FUNCTION_BLOCK FB_AlarmControler EXTENDS FB_VisuEventsHandling IMPLEMENTS I_AlarmControler
VAR
	sName 					: STRING;					(*  *)

	bInit 					: BOOL;						(*  *)
	bAbort 					: BOOL;						(*  *)
	bClear					: BOOL;						(*  *)
	bClearAll 				: BOOL;						(*  *)
	bConfirm 				: BOOL;						(*  *)
	bConfirmAll 			: BOOL;						(*  *)
	bExport 				: BOOL;						(*  *)
	
	bResetConfirmation 		: BOOL;						(*  *)
	sFileName				: STRING;					(*  *)
	
	bActive 				: BOOL;						(*  *)
	bBusy					: BOOL;						(*  *)
	bError					: BOOL;						(*  *)
	iErrorID 				: HRESULT;					(*  *)
	iResult					: HRESULT;					(*  *)
	eAlarmControlerState 	: E_AlarmControlerState;	(*  *)
	
	ipFilter 				: I_TcEventFilter;			(*  *)
	fbEventLogger 			: FB_TcEventLogger;			(*  *)
END_VAR

(* Execute parent logic *)
SUPER^();

(* Run main state machine *)
StateMachine();

PROPERTY Active : REFERENCE TO BOOL
GET
Active REF= bActive;
END_GET
END_PROPERTY

PROPERTY ActiveCritical : REFERENCE TO UDINT
GET
ActiveCritical REF= iActiveCritical;
END_GET
END_PROPERTY

PROPERTY ActiveError : REFERENCE TO UDINT
GET
ActiveError REF= iActiveError;
END_GET
END_PROPERTY

PROPERTY ActiveInfo : REFERENCE TO UDINT
GET
ActiveInfo REF= iActiveInfo;
END_GET
END_PROPERTY

PROPERTY ActiveVerbose : REFERENCE TO UDINT
GET
ActiveVerbose REF= iActiveVerbose;
END_GET
END_PROPERTY

PROPERTY ActiveWarrning : REFERENCE TO UDINT
GET
ActiveWarrning REF= iActiveWarning;
END_GET
END_PROPERTY

PROPERTY AlarmsTable : REFERENCE TO ARRAY[1..iMAX_EVENTS] OF ST_Event
GET
AlarmsTable REF= arrActiveAlarms;
END_GET
END_PROPERTY

PROPERTY Busy : REFERENCE TO BOOL
GET
Busy REF= bBusy;
END_GET
END_PROPERTY

PROPERTY Error : REFERENCE TO BOOL
GET
Error REF= bError;
END_GET
END_PROPERTY

PROPERTY ErrorID : REFERENCE TO HRESULT
GET
ErrorID REF= iResult;
END_GET
END_PROPERTY

PROPERTY EventsTable : REFERENCE TO ARRAY[1..iMAX_EVENTS] OF ST_Event
GET
EventsTable REF= arrEvents;
END_GET
END_PROPERTY

PROPERTY FileName : STRING
GET
FileName := sFileName;
END_GET
SET
sFileName := FileName;
END_SET
END_PROPERTY

PROPERTY MaxEvents : UDINT
GET
MaxEvents := iMAX_EVENTS;
END_GET
END_PROPERTY

METHOD MR_Abort : BOOL
VAR_INPUT
END_VAR
IF eAlarmControlerState > ALARM_CONTROLER_UNINITIALIZED THEN
	bAbort := TRUE;
	MR_Abort := FALSE;
	bBusy := TRUE;
	
	eAlarmControlerState := ALARM_CONTROLER_ABORTING;
	fbMachineLogger.MR_AddLogs(CONCAT(sName,' : abort requested'));	
	
ELSIF eAlarmControlerState = ALARM_CONTROLER_UNINITIALIZED THEN
	bAbort := FALSE;
	MR_Abort := TRUE;
	bBusy := FALSE;
	bActive := FALSE;
	
	fbMachineLogger.MR_AddLogs(CONCAT(sName,' : abort done'));	
	
END_IF
END_METHOD

METHOD MR_Clear : BOOL
VAR_INPUT
	ipFilter : I_TcEventFilter;
	bResetConfirmation : BOOL;
END_VAR
IF eAlarmControlerState = ALARM_CONTROLER_IDLE THEN
	bClear := TRUE;
	MR_Clear := FALSE;
	bBusy := TRUE;
	THIS^.ipFilter := ipFilter;
	THIS^.bResetConfirmation := bResetConfirmation;
	
	eAlarmControlerState := ALARM_CONTROLER_CLEAR;
	fbMachineLogger.MR_AddLogs(CONCAT(sName,' : clear requested'));		
	
ELSIF eAlarmControlerState = ALARM_CONTROLER_CLEAR_DONE THEN
	bClear := FALSE;
	MR_Clear := TRUE;	
	bBusy := FALSE;
	
	fbMachineLogger.MR_AddLogs(CONCAT(sName,' : clear done'));		
	
END_IF
END_METHOD

METHOD MR_ClearAll : BOOL
VAR_INPUT
	bResetConfirmation : BOOL;
END_VAR
IF eAlarmControlerState = ALARM_CONTROLER_IDLE THEN
	bClearAll := TRUE;
	MR_ClearAll := FALSE;
	bBusy := TRUE;
	THIS^.bResetConfirmation := bResetConfirmation;
	
	eAlarmControlerState := ALARM_CONTROLER_CLEAR_ALL;
	fbMachineLogger.MR_AddLogs(CONCAT(sName,' : clear all requested'));		

ELSIF eAlarmControlerState = ALARM_CONTROLER_CLEAR_ALL_DONE THEN
	bClearAll := FALSE;
	MR_ClearAll := TRUE;
	bBusy := FALSE;
	
	fbMachineLogger.MR_AddLogs(CONCAT(sName,' : clear all done'));		
	
END_IF
END_METHOD

METHOD MR_Confirm : BOOL
VAR_INPUT
	ipFilter : I_TcEventFilter;
END_VAR
IF eAlarmControlerState = ALARM_CONTROLER_IDLE THEN
	bConfirm := TRUE;
	MR_Confirm := FALSE;
	bBusy := TRUE;
	THIS^.ipFilter := ipFilter;
	
	eAlarmControlerState := ALARM_CONTROLER_CONFIRM;
	fbMachineLogger.MR_AddLogs(CONCAT(sName,' : confirmation requested'));		
	
ELSIF eAlarmControlerState = ALARM_CONTROLER_CONFIRM_DONE THEN
	bConfirm := FALSE;
	MR_Confirm := TRUE;	
	bBusy := FALSE;
	
	fbMachineLogger.MR_AddLogs(CONCAT(sName,' : confirmation done'));		
	
END_IF
END_METHOD

METHOD MR_ConfirmAll : BOOL
VAR_INPUT
	bResetConfirmation : BOOL;
END_VAR
IF eAlarmControlerState = ALARM_CONTROLER_IDLE THEN
	bConfirmAll := TRUE;
	MR_ConfirmAll := FALSE;
	bBusy := TRUE;
	
	THIS^.bResetConfirmation := bResetConfirmation;
	eAlarmControlerState := ALARM_CONTROLER_CONFIRM_ALL;
	fbMachineLogger.MR_AddLogs(CONCAT(sName,' : confirmation of all requested'));		
	
ELSIF eAlarmControlerState = ALARM_CONTROLER_CONFIRM_ALL_DONE THEN
	bConfirmAll := FALSE;
	MR_ConfirmAll := TRUE;
	bBusy := FALSE;
	
	fbMachineLogger.MR_AddLogs(CONCAT(sName,' : confirmation of all done'));	
	
END_IF
END_METHOD

METHOD MR_Export : BOOL
VAR_INPUT
END_VAR
IF eAlarmControlerState = ALARM_CONTROLER_IDLE THEN
	bExport := TRUE;
	MR_Export := FALSE;
	bBusy := TRUE;
	
	eAlarmControlerState := ALARM_CONTROLER_EXPORT;
	fbMachineLogger.MR_AddLogs(CONCAT(sName,' : exportation requested'));	
	
ELSIF eAlarmControlerState = ALARM_CONTROLER_EXPORT_DONE THEN
	bExport := FALSE;
	MR_Export := TRUE;
	bBusy := FALSE;
	
	fbMachineLogger.MR_AddLogs(CONCAT(sName,' : exportation done'));	
	
END_IF
END_METHOD

METHOD MR_FirstCycle : BOOL
VAR_INPUT
	sName 		: STRING;
	sFileName 	: STRING;
END_VAR
THIS^.sName := sName;
THIS^.sFileName := sFileName;
END_METHOD

METHOD MR_Init : BOOL
VAR_INPUT
END_VAR
IF eAlarmControlerState = ALARM_CONTROLER_UNINITIALIZED THEN
	MR_Init := FALSE;
	bInit := TRUE;
	bBusy := TRUE;
	
	eAlarmControlerState := ALARM_CONTROLER_INITIALIZING;
	fbMachineLogger.MR_AddLogs(CONCAT(sName,' : initialization requested'));
	
ELSIF eAlarmControlerState = ALARM_CONTROLER_IDLE THEN
	bInit := FALSE;
	MR_Init := FALSE;
	bBusy := FALSE;
	bActive := TRUE;
	
	fbMachineLogger.MR_AddLogs(CONCAT(sName,' : initialization done'));
	
END_IF
END_METHOD

METHOD PROTECTED MS_Aborting
VAR_INPUT
END_VAR
Unsubscribe();
eAlarmControlerState := ALARM_CONTROLER_UNINITIALIZED;
END_METHOD

METHOD PROTECTED MS_Clear
VAR_INPUT
END_VAR
fbEventLogger.ConfirmAllAlarms(	nTimeStamp := 0);

iResult := fbEventLogger.ClearAlarms(	nTimeStamp 			:= 0,
										bResetConfirmation	:= bResetConfirmation,
										ipFilter 			:= ipFilter);

IF iResult = S_OK THEN
	eAlarmControlerState := ALARM_CONTROLER_CLEAR_DONE;
END_IF
END_METHOD

METHOD PROTECTED MS_ClearAll
VAR_INPUT
END_VAR
fbEventLogger.ConfirmAllAlarms(	nTimeStamp := 0);

iResult := fbEventLogger.ClearAllAlarms(	nTimeStamp := 0,
											bResetConfirmation := bResetConfirmation);

IF iResult = S_OK THEN
	eAlarmControlerState := ALARM_CONTROLER_CLEAR_ALL_DONE;
END_IF
END_METHOD

METHOD PROTECTED MS_ClearAllDone
VAR_INPUT
END_VAR
IF NOT bClearAll THEN
	eAlarmControlerState := ALARM_CONTROLER_IDLE;
END_IF
END_METHOD

METHOD PROTECTED MS_ClearDone
VAR_INPUT
END_VAR
IF NOT bClear THEN
	eAlarmControlerState := ALARM_CONTROLER_IDLE;
END_IF
END_METHOD

METHOD PROTECTED MS_Confirm
VAR_INPUT
END_VAR
iResult := fbEventLogger.ConfirmAlarms(	nTimeStamp	:= 0,
										ipFilter	:= ipFilter); 
										
IF iResult = S_OK THEN
	eAlarmControlerState := ALARM_CONTROLER_CONFIRM_DONE;
END_IF
END_METHOD

METHOD PROTECTED MS_ConfirmAll
VAR_INPUT
END_VAR
fbEventLogger.ConfirmAllAlarms(	nTimeStamp := 0);

iResult := fbEventLogger.ClearAllAlarms(	nTimeStamp := 0,
											bResetConfirmation := bResetConfirmation);
	
IF iResult = S_OK THEN
	eAlarmControlerState := ALARM_CONTROLER_CONFIRM_ALL_DONE;
END_IF
END_METHOD

METHOD PROTECTED MS_ConfirmAllDone
VAR_INPUT
END_VAR
IF NOT bConfirmAll THEN
	eAlarmControlerState := ALARM_CONTROLER_IDLE;
END_IF
END_METHOD

METHOD PROTECTED MS_ConfirmDone
VAR_INPUT
END_VAR
IF NOT bConfirm THEN
	eAlarmControlerState := ALARM_CONTROLER_IDLE;
END_IF
END_METHOD

METHOD PROTECTED MS_Export
VAR_INPUT
END_VAR
fbEventLogger.ExportLoggedEvents( 	sFileName := sFileName,
									ipExportSettings := 0,
									bError => bError,
									hrErrorCode => iResult);

IF iResult = S_OK THEN
	eAlarmControlerState := ALARM_CONTROLER_EXPORT_DONE;
END_IF
END_METHOD

METHOD PROTECTED MS_ExportDone
VAR_INPUT
END_VAR
IF NOT bExport THEN
	eAlarmControlerState := ALARM_CONTROLER_IDLE;
END_IF
END_METHOD

METHOD PROTECTED MS_Idle
VAR_INPUT
END_VAR
;
END_METHOD

METHOD PROTECTED MS_Initializing
VAR_INPUT
END_VAR
Subscribe(0, 0);
eAlarmControlerState := ALARM_CONTROLER_READY_INITIALIZED;
END_METHOD

METHOD PROTECTED MS_ReadyInitialized
VAR_INPUT
END_VAR
bActive := TRUE;
eAlarmControlerState := ALARM_CONTROLER_IDLE;
END_METHOD

METHOD PROTECTED MS_Uninitialized
VAR_INPUT
END_VAR
bActive := FALSE;
END_METHOD

PROPERTY Name : REFERENCE TO STRING
GET
Name REF= sName;
END_GET
END_PROPERTY

PROPERTY State : REFERENCE TO E_AlarmControlerState
GET
State REF= eAlarmControlerState;
END_GET
END_PROPERTY

METHOD PROTECTED StateMachine
VAR_INPUT
END_VAR
CASE eAlarmControlerState OF
	ALARM_CONTROLER_UNINITIALIZED:
		MS_Uninitialized();
	
	ALARM_CONTROLER_INITIALIZING:
		MS_Initializing();
		
	ALARM_CONTROLER_READY_INITIALIZED:
		MS_ReadyInitialized();	
	
	ALARM_CONTROLER_IDLE:
		MS_Idle();
		
	ALARM_CONTROLER_CONFIRM_ALL:
		MS_ConfirmAll();
		
	ALARM_CONTROLER_CONFIRM_ALL_DONE:
		MS_ConfirmAllDone();
	
	ALARM_CONTROLER_CLEAR_ALL:
		MS_ClearAll();
		
	ALARM_CONTROLER_CLEAR_ALL_DONE:
		MS_ClearAllDone();
		
	ALARM_CONTROLER_CONFIRM:
		MS_Confirm();
	
	ALARM_CONTROLER_CONFIRM_DONE:
		MS_ConfirmDone();
		
	ALARM_CONTROLER_CLEAR:
		MS_Clear();
		
	ALARM_CONTROLER_CLEAR_DONE:
		MS_ClearDone();
		
	ALARM_CONTROLER_EXPORT:
		MS_Export();
		
	ALARM_CONTROLER_EXPORT_DONE:
		MS_ExportDone();
		
	ALARM_CONTROLER_ABORTING:
		MS_Aborting();
		
END_CASE
END_METHOD

END_FUNCTION_BLOCK

(* stored: Version 1.1.0.1, ProductVersion 3.1.4024.12
   POU FB_AlarmControler: Id {ddec5e34-e3bc-45f8-b972-1b6ce9bbff8e}, SpecialFunc None
   Folder FirstCycle: Id {1deae082-c280-4c73-bdbd-1c727dd4349b}
   Folder Properties: Id {8baaa26c-c607-4a0d-a497-996b10dc2f95}
   Folder Parameters: Id {ef59bcca-49b8-4d4d-989a-3f54a795c26a}
   Folder Status: Id {373f4e82-d21e-4eb3-9d14-ffccd0b59498}
   Folder Requests: Id {b07a92d9-40cc-41fe-9d19-612b76cd42ed}
   Folder StateMachine: Id {c34d18ca-e3a2-426d-9d95-b99fdadf1226}
   Property Active: Id {e95ca6c6-abc5-4a91-9c2d-ddc238665bd2}
   Get Get: Id {31069402-77c6-4971-a5e7-4777b2a7f017}
   Property ActiveCritical: Id {4141f6dd-928b-41fc-b531-033fb127c1ce}
   Get Get: Id {b8674030-a376-474d-aa7e-aea9dce4974e}
   Property ActiveError: Id {f1bb7335-2627-49c3-b32e-4f10ad21b069}
   Get Get: Id {8354ae32-3f51-4088-ace4-f33a84174ee0}
   Property ActiveInfo: Id {2756b7a4-47c5-47b4-b542-e6c23e6ace7b}
   Get Get: Id {a00edf67-e751-4d4c-8955-99249838d0ae}
   Property ActiveVerbose: Id {0c82e7fd-831f-4698-9b25-7119d89d3902}
   Get Get: Id {e34d361a-9a10-4dd0-b9a5-9e81508ad3fc}
   Property ActiveWarrning: Id {894dc690-3b3a-41d1-bb2e-6dbb63394eef}
   Get Get: Id {be527dfb-1012-4c2e-8940-ff2abf4dbaba}
   Property AlarmsTable: Id {9a0a0be8-e15c-4c01-b09f-2a5c72a8d50f}
   Get Get: Id {3d9a68e7-85f5-4ba1-a280-17a34bbbba4d}
   Property Busy: Id {aaf05382-2f29-4190-82e2-502d4a3f302b}
   Get Get: Id {296a7e49-0717-4e9e-bff4-5a7eeeb7cc6b}
   Property Error: Id {ceab45ad-3baa-46ca-ace7-04ad0413c221}
   Get Get: Id {d0db2535-cf60-4569-84b3-7c8ad6331d16}
   Property ErrorID: Id {892bfa99-5240-43ae-9041-c383011cf26e}
   Get Get: Id {172f8216-04b4-47b6-bc64-636af9f20d92}
   Property EventsTable: Id {dedb517f-f504-4aef-b70d-e2471d1a6337}
   Get Get: Id {9e580b70-defb-4a1e-9baa-c58786e4b12f}
   Property FileName: Id {2c7867ab-37bd-447c-8628-759fcbc21ed8}
   Get Get: Id {31ede752-443e-4a94-8502-ba92f68bb2ef}
   Set Set: Id {1f40f16b-815b-4e24-82ae-54238f7002c2}
   Property MaxEvents: Id {8870cc92-bae7-418a-9b6a-a769efae540d}
   Get Get: Id {1120577d-ddbf-4311-9719-9784288c9207}
   Method MR_Abort: Id {fc60768f-5a43-451c-9f41-b2b9cc000fa0}
   Method MR_Clear: Id {dc077892-7b8c-4259-a8bf-59a165666697}
   Method MR_ClearAll: Id {ca3d95ac-c22b-4241-ade4-cf38d48a98c7}
   Method MR_Confirm: Id {2ff78302-1725-44d8-820f-f9bc5a758d1e}
   Method MR_ConfirmAll: Id {b8270bbf-43ac-4be6-92f6-32353a97dfa5}
   Method MR_Export: Id {d859110a-3929-4202-847d-3672d1159e4b}
   Method MR_FirstCycle: Id {a8bb1a3b-eb56-4c2d-9e59-27555d0c90c5}
   Method MR_Init: Id {da33a874-b294-4d56-9212-e42bfc2800c8}
   Method MS_Aborting: Id {fb96b0e3-e321-4a44-85d7-9c2cf91a02ba}
   Method MS_Clear: Id {520a997e-b6a3-40db-bf4b-b7170e843dd1}
   Method MS_ClearAll: Id {e81af08a-dfdd-4d2f-ba36-7efe39bf640b}
   Method MS_ClearAllDone: Id {0b3d4170-e6c2-41f8-8048-6f0ac533e6bf}
   Method MS_ClearDone: Id {e4ae38e5-600a-4580-8e5c-5e20a1482367}
   Method MS_Confirm: Id {2a91952f-e147-426c-b8f0-acd0676f4b8a}
   Method MS_ConfirmAll: Id {c079069d-c5af-43b8-adcc-88a2a73fa838}
   Method MS_ConfirmAllDone: Id {32f9f854-2aa4-43d5-a627-d990f08a4914}
   Method MS_ConfirmDone: Id {37eab967-9c5d-447d-b83c-3ce8b956d3c4}
   Method MS_Export: Id {a06d2090-2c3f-4571-85c5-ff405d7dc2e6}
   Method MS_ExportDone: Id {fca97323-c328-4411-8a74-0c09b795da4e}
   Method MS_Idle: Id {b60488f3-5515-4b06-9ce0-64be9315b129}
   Method MS_Initializing: Id {019f0877-7a74-43b0-a683-3b3650abd43b}
   Method MS_ReadyInitialized: Id {caedb33e-e010-444a-a577-e58d80059496}
   Method MS_Uninitialized: Id {df8b0f15-446f-4062-ba8d-389ad85d080d}
   Property Name: Id {ccb33e78-e893-4925-95c0-5e72758fa8d7}
   Get Get: Id {579e0bcf-bcf3-4317-98fb-723d1235815e}
   Property State: Id {e064c1d6-466f-4b19-9b4c-43d3580347cb}
   Get Get: Id {0c06a4f5-2f50-4d42-9fdb-962bf8bd5620}
   Method StateMachine: Id {3441ea60-6baf-4178-97c5-15a56c893a55} *)
